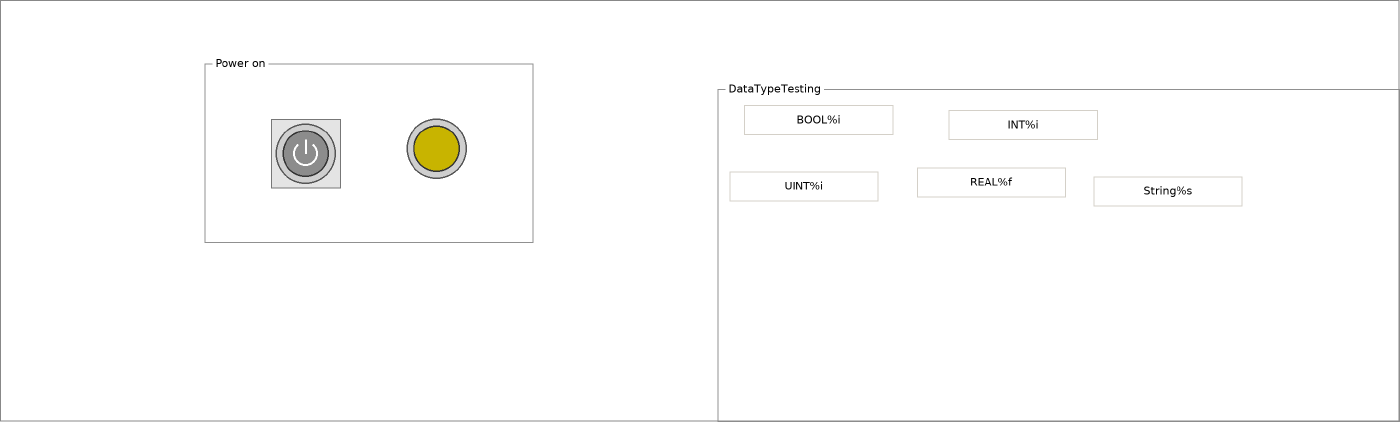
VISUALIZATION HMI  // 1411x426
    GroupBox (206,56 331x189), "Power on"
        PowerSwitch (67,64 70x70), variable: MAIN.bStart, behaviour: TOGGLE, style: Switch-PowerSwitch-Gray
        Lamp1 (199,59 70x70), variable: MAIN.bEnable, style: Lamp-Lamp1-Yellow
    GroupBox (723,82 688x344), "DataTypeTesting"
        Textfield (27,24 150x30), "BOOL%i", text variable: MAIN.bEnable
        Textfield (233,29 150x30), "INT%i", text variable: MAIN.nInt
        Textfield (12,91 150x30), "UINT%i", text variable: MAIN.nUINT
        Textfield (201,87 150x30), "REAL%f", text variable: MAIN.fREAL
            OnMouseDown: write the text variable via Default
        Textfield (379,96 150x30), "String%s", text variable: MAIN.sPowerStatus
            OnMouseDown: write the text variable via Default
END_VISUALIZATION

(* stored: Version 1.1.0.1, ProductVersion 3.1.4024.12
   Visu HMI: Id {e3f2f2fa-798b-43ff-a021-ac26d6589e0a} *)
